# EPICS StreamDevice protocol: protocol/data.proto
OutTerminator = LF;
ReplyTimeout = 1000;
ReadTimeout  = 100;
InTerminator = LF;

read_adc {
	Separator     = "";
	InTerminator  = "";
	out "ADC %(\$1.VAL)d";
	in  "%d\n";
}
